// TwinCAT 3 PLC project cpu
// ProgramVersion: 3.1.4024.0
// libraries:
//   p6lib_common, * (MacGregor)
//   Tc2_Standard, * (Beckhoff Automation GmbH)
//   Tc2_System, * (Beckhoff Automation GmbH)
//   Tc3_Module, * (Beckhoff Automation GmbH)
// project tree:
//   GVLs/ Alarms.TcGVL, counters.TcGVL, gvlMisc.TcGVL
//   / MAIN.TcPOU, PlcTask.TcTTO
//   POUs/ counter.TcPOU, makeAlarm.TcPOU

CONFIGURATION cpu
    RESOURCE PLC ON TwinCAT3
        TASK PlcTask(INTERVAL := T#10ms, PRIORITY := 20);
        PROGRAM MAIN WITH PlcTask : MAIN;
    END_RESOURCE
END_CONFIGURATION

// ---- GVLs/Alarms.TcGVL
{attribute 'qualified_only'}
VAR_GLOBAL
	
    p6alarm1		: p6com.AlarmDigital(TC_Events.Alarms.Alarm1);
	p6alarm2		: p6com.AlarmDigital(TC_Events.Alarms.Alarm2);
    
    alarm1 : makeAlarm(alarm:=p6alarm1, onTime:=T#5.5S, offTime:=T#10S);
    alarm2 : makeAlarm(alarm:=p6alarm2, onTime:=T#22.5S, offTime:=T#30S);
    
END_VAR

// ---- GVLs/counters.TcGVL
{attribute 'qualified_only'}
VAR_GLOBAL
    counter01 : counter(23);
    counter02 : counter(2);
    counter03 : counter(233);
    counter04 : counter(2);
    counter05 : counter(27);
    counter06 : counter(21);
    counter07 : counter(55);
    counter08 : counter(67);
    counter09 : counter(10);
    counter10 : counter(98);
    counter11 : counter(666);
    counter12 : counter(999);
    counter13 : counter(1000);
    counter14 : counter(333);
    counter15 : counter(445);
    counter16 : counter(4454089);
    counter17 : counter(56464569);
    counter18 : counter(098402423);
    counter19 : counter(33355);
    counter20 : counter(93783);

    numbers : ARRAY[0..199] OF DINT;
    
END_VAR

// ---- GVLs/gvlMisc.TcGVL
{attribute 'qualified_only'}
VAR_GLOBAL
    data01 : DINT;
    data02 : DINT;
    data03 : DINT;
    data04 : DINT;
END_VAR

// ---- MAIN.TcPOU
PROGRAM MAIN
VAR
    value : DINT; 
    timer : TON;
END_VAR

timer(IN:= NOT timer.Q, PT:=T#80MS);

//Alarms.alarm1();
//Alarms.alarm2();


counters.counter01();
counters.counter02();
counters.counter03();
counters.counter04();
counters.counter05();
counters.counter06();
counters.counter07();
counters.counter08();
counters.counter09();
counters.counter10();
counters.counter11();
counters.counter12();
counters.counter13();
counters.counter14();
counters.counter15();
counters.counter16();
counters.counter17();
counters.counter18();
counters.counter19();
counters.counter20();


value := counters.counter01.Value;
value := counters.counter02.Value;
value := counters.counter03.Value;
value := counters.counter04.Value;
value := counters.counter05.Value;
value := counters.counter06.Value;
value := counters.counter07.Value;
value := counters.counter08.Value;
value := counters.counter09.Value;
value := counters.counter10.Value;
value := counters.counter11.Value;
value := counters.counter12.Value;
value := counters.counter13.Value;
value := counters.counter14.Value;
value := counters.counter15.Value;
value := counters.counter16.Value;
value := counters.counter17.Value;
value := counters.counter18.Value;
value := counters.counter19.Value;
value := counters.counter20.Value;

END_PROGRAM

// ---- POUs/makeAlarm.TcPOU
FUNCTION_BLOCK makeAlarm
VAR
    alarm : REFERENCE TO p6com.AlarmDigital;
    onTime : TIME;
    offTime : TIME;

    onTimer : TON; 
    offTimer: TON;
    state : DINT;
 
END_VAR



onTimer(IN:= state=0, PT:= onTime);
offTimer(IN:= state=10, PT:= offTime);

CASE state OF
    0: 
        IF onTimer.Q THEN
            state := 10;
		END_IF
        
    10:
        IF offTimer.Q THEN
            state := 0;
		END_IF
END_CASE

alarm(ID:=2, IDName:='Alarm 1', Value := state = 10, TimeSpan := T#1MS);

METHOD FB_init : BOOL
VAR_INPUT
	bInitRetains : BOOL; // if TRUE, the retain variables are initialized (warm start / cold start)
	bInCopyCode : BOOL;  // if TRUE, the instance afterwards gets moved into the copy code (online change)
    alarm : REFERENCE TO p6com.AlarmDigital;
    onTime : TIME;
    offTime : TIME;
END_VAR
THIS^.alarm REF= alarm;
THIS^.onTime := onTime;
THIS^.offTime := offTime;
END_METHOD

END_FUNCTION_BLOCK

// ---- POUs/counter.TcPOU
FUNCTION_BLOCK counter
VAR
    counter : DINT; 
END_VAR

counter := counter + 1;

METHOD FB_init : BOOL
VAR_INPUT
	bInitRetains : BOOL; // if TRUE, the retain variables are initialized (warm start / cold start)
	bInCopyCode : BOOL;  // if TRUE, the instance afterwards gets moved into the copy code (online change)
    start : DINT;
END_VAR
counter := start;
END_METHOD

{attribute 'monitoring' := 'call'}
{attribute 'TcRpcEnable'}
PROPERTY Value : DINT
GET
Value := THIS^.counter;
END_GET
SET
THIS^.counter := Value;
END_SET
END_PROPERTY

END_FUNCTION_BLOCK
